// TIA Portal V17 export
// export: Created 2021-11-24T11:00:24.876193Z, ExportSetting WithDefaults, DisplayName Totally Integrated Automation Portal, DisplayVersion V17, DisplayName TIA Portal Openness, DisplayVersion V17, DisplayName TIA Portal Version Control Interface, DisplayVersion V17, DisplayName SINAMICS Startdrive Advanced, DisplayVersion V17, DisplayName SINAMICS Startdrive G130, G150, S120, S150, SINAMICS MV, S210, DisplayVersion V17, DisplayName SINAMICS Startdrive G110M, G120, G120C, G120D, G120P, G115D, DisplayVersion V17, DisplayName STEP 7 Professional, DisplayVersion V17, DisplayName STEP 7 Safety, DisplayVersion V17, DisplayName WinCC Advanced / Unified PC, DisplayVersion V17
VAR_GLOBAL   // PLC tag table "Default tag table"
   vystup2 AT %Q1.0 : Bool;
   vystup1 AT %Q0.0 : Bool;
   Tag_1 AT %MW50 : Int;
   Tag_2 AT %MW52 : Word;
   Tag_3 AT %MW54 : Int;
   Tag_4 AT %MW56 : Word;
   vstup2 AT %I20.0 : Bool;
   vstup1 AT %I20.1 : Bool;
   xxx AT %I20.2 : Bool;
END_VAR
